// TIA Portal V19 export
DATA_BLOCK "DB_PNOZ_Receive"   // DB364
{ S7_Optimized_Access := 'FALSE' }
// stored: AutoNumber false
   VAR
      In : Struct
         Header : Array[0..7] of Byte;
         VirtualInput : Array[0..127] of Bool;
         LED_0_Fault : Bool;   // LED 0 Fault
         LED_1_Fault : Bool;   // LED 1 Fault
         LED_Fault : Bool;   // LED Fault
         LED_Diag : Bool;   // LED Diag
         LED_Run_ST : Bool := false;   // LED Run
         reserved1 : Bool;   // reserved
         LED_Run_FS : Bool := false;   // reserved
         Data_cons_check_bit : Bool;   // Data consistence check bit
         Table_Nr : Byte;   // Table Nr
         Segment : Struct
            Nr : Byte;
            Byte_0 : Byte;
            Byte_1 : Byte;
            Byte_2 : Byte;
            Byte_3 : Byte;
            Byte_4 : Byte;
            Byte_5 : Byte;
            Byte_6 : Byte;
            Byte_7 : Byte;
            Byte_8 : Byte;
            Byte_9 : Byte;
            Byte_10 : Byte;
            Byte_11 : Byte;
            Byte_12 : Byte;
         END_STRUCT;
         reserviert : Byte;
         Checksum : Byte := BYTE#16#0;   // Checksumme, Byte 4 + Byte 39
         Endekennung : Byte := BYTE#16#10;   // last Byte, must be 0x10 every time!
      END_STRUCT;
   END_VAR
BEGIN
   In.Header[0] := BYTE#16#05;
   In.Header[1] := BYTE#16#15;
   In.Header[3] := BYTE#16#26;
   In.Header[4] := BYTE#16#DC;
   In.VirtualInput[0] := TRUE;
   In.VirtualInput[18..23] := TRUE;
   In.VirtualInput[35..36] := TRUE;
END_DATA_BLOCK
